// TIA Portal V17 export
// export: Created 2026-04-13T11:12:42.5502863Z, ExportSetting WithDefaults, DisplayName Totally Integrated Automation Portal, DisplayVersion V17 Update 4, DisplayName TIA Portal Openness, DisplayVersion V17 Update 4, DisplayName TIA Portal Version Control Interface, DisplayVersion V17, DisplayName SINAMICS Startdrive Advanced, DisplayVersion V17, DisplayName SINAMICS Startdrive G130, G150, S120, S150, SINAMICS MV, S210, DisplayVersion V17, DisplayName SINAMICS Startdrive G110M, G120, G120C, G120D, G120P, G115D, DisplayVersion V17, DisplayName STEP 7 Professional, DisplayVersion V17 Update 4, DisplayName STEP 7 Safety, DisplayVersion V17, DisplayName WinCC Professional, DisplayVersion V17 Update 4
FUNCTION_BLOCK "0-模拟量输入1PID"   // FB172, LAD
{ S7_Optimized_Access := 'TRUE' }
VERSION : 0.1
// stored: AutoNumber true, IsIECCheckEnabled false, IsRetainMemResEnabled false, MemoryReserve 100, SetENOAutomatically false, UDAEnableTagReadback false
   VAR_INPUT
      "仪表反馈值(模拟量)" : Int;
      积分P : Real := 0.5;
      微分I : Real := 0.5;
      "上限(模拟量)" : Real := 27648.0;
      "下限(模拟量)" : Real;
      "上限(工程量)" : Real := 200.0;
      "下限(工程量)" : Real;
      "设定补偿值(工程量)" : Real := 0.5;   // PID值快到达设定值时由于PID调节作用始终差一点才能到达设定值，所以用补偿的方式直接加上
      "设定目标值(工程量)" : Real := 100.0;
   END_VAR
   VAR_OUTPUT
      "仪表反馈值(工程量)" : Real;   // 由模拟量输入直接比例缩放转出的工程量，作用就是看一下显示
      "给定变频器(模拟量)" : Int;   // PID调节后的直接给变频器的模拟量值0-27648
      "PID调节输出值(工程量)" : Real;
   END_VAR
   VAR
      临时模拟量数据输入 : Real;
      缩放比例 : Real;
      实际模拟量 : Real;
      当前偏差 : Real;
      上一次偏差 : Real;
      输出控制量 : Real;
      PQW : Real;
   END_VAR
BEGIN

REGION Network 1 (SCL)
   //模拟量转换工程值
   #临时模拟量数据输入 := INT_TO_REAL(#"仪表反馈值(模拟量)");  //将模拟量输入转换为real类型
   #缩放比例 := (#"上限(工程量)" - #"下限(工程量)") / (#"上限(模拟量)" - #"下限(模拟量)");//算出实际值与模拟量的缩放比例
   #"仪表反馈值(工程量)" := (#"仪表反馈值(模拟量)"-#"下限(模拟量)") * #缩放比例+#"下限(工程量)";      //转换完成
   #当前偏差 := #"设定目标值(工程量)" - #"仪表反馈值(工程量)";

   //PID计算
   IF  #"设定补偿值(工程量)">ABS( #当前偏差) THEN
       #输出控制量 := 0;
   ELSIF #"设定补偿值(工程量)"<ABS( #当前偏差) THEN
       #输出控制量 := #积分P*(#当前偏差-#上一次偏差)+#微分I*#当前偏差;
   END_IF;

   #"PID调节输出值(工程量)":=#输出控制量;

   //上下限制
   IF #"PID调节输出值(工程量)"> #"上限(工程量)"THEN
       #"PID调节输出值(工程量)" := #"上限(工程量)";
   ELSIF #"PID调节输出值(工程量)"< #"下限(工程量)"THEN
       #"PID调节输出值(工程量)" := #"下限(工程量)";
   END_IF;


   //控制电机输出

   #上一次偏差 := #当前偏差;
   #PQW:=(#"PID调节输出值(工程量)"-#"下限(工程量)")/(#"上限(工程量)"-#"下限(工程量)")*#"上限(模拟量)";
   #"给定变频器(模拟量)" := REAL_TO_INT(#PQW);
END_REGION
END_FUNCTION_BLOCK
